{attribute 'linkalways'} 
{attribute 'no_explicit_call' := 'This FB is a CLASS and must be accessed using methods or properties'}
{attribute 'enable_dynamic_creation'}
FUNCTION_BLOCK _ETcVnDistanceType EXTENDS EnumDatatypeBase
VAR
	localData : ETcVnDistanceType;
	activeData : REFERENCE TO ETcVnDistanceType;
	enumBaseDatatype : _DINT(localData);
END_VAR

METHOD PRIVATE AddLocalEnumeration
VAR_INPUT
	Enumeration : T_MAXSTRING;
	Value : ETcVnDistanceType;
END_VAR
AddEnumeration(Enumeration, Value);
END_METHOD

PROPERTY PUBLIC Address : PVOID
GET
Address := ADR(activeData);
END_GET
END_PROPERTY

METHOD PUBLIC ClearReference
VAR_INPUT
END_VAR
activeData REF= localData;
SetBaseDatatypeReference();
END_METHOD

METHOD PUBLIC Clone : I_Datatype
VAR
    pClone : POINTER TO _ETcVnDistanceType;
END_VAR
pClone := __NEW(_ETcVnDistanceType(InitialValue := Value));
Clone := pClone^;
END_METHOD

METHOD FB_init : BOOL
VAR_INPUT
	bInitRetains : BOOL; // if TRUE, the retain variables are initialized (warm start / cold start)
	bInCopyCode : BOOL;  // if TRUE, the instance afterwards gets moved into the copy code (online change)
	InitialValue : ETcVnDistanceType;
END_VAR
localData := InitialValue;
AddBaseDatatype(enumBaseDatatype);
ClearReference();

AddLocalEnumeration('TCVN_DT_USER', ETcVnDistanceType.TCVN_DT_USER);
AddLocalEnumeration('TCVN_DT_L1', ETcVnDistanceType.TCVN_DT_L1);
AddLocalEnumeration('TCVN_DT_L2', ETcVnDistanceType.TCVN_DT_L2);
AddLocalEnumeration('TCVN_DT_C', ETcVnDistanceType.TCVN_DT_C);
AddLocalEnumeration('TCVN_DT_L12', ETcVnDistanceType.TCVN_DT_L12);
AddLocalEnumeration('TCVN_DT_FAIR', ETcVnDistanceType.TCVN_DT_FAIR);
AddLocalEnumeration('TCVN_DT_WELSCH', ETcVnDistanceType.TCVN_DT_WELSCH);
AddLocalEnumeration('TCVN_DT_HUBER ', ETcVnDistanceType.TCVN_DT_HUBER);
END_METHOD

PROPERTY PUBLIC Identifier : T_MAXSTRING
GET
Identifier := 'ETcVnDistanceType';
END_GET
END_PROPERTY

METHOD IsEnumeratorValueEqual : BOOL
VAR_INPUT
	Enumerator : I_KeyValueForwardEnumerator;
END_VAR
VAR
	storedValue : ETcVnDistanceType;
END_VAR
IF NOT Enumerator.TryGet(storedValue) THEN
	RETURN;
END_IF

IsEnumeratorValueEqual := storedValue = activeData;
END_METHOD

METHOD PUBLIC MakeReferenceTo
VAR_INPUT
	ReferenceTarget : REFERENCE TO ETcVnDistanceType;
END_VAR
activeData REF= ReferenceTarget;
SetBaseDatatypeReference();
END_METHOD

METHOD PROTECTED SetBaseDatatypeReference
VAR_INPUT
END_VAR
enumBaseDatatype.MakeReferenceTo(activeData);
END_METHOD

PROPERTY PUBLIC Size : UDINT
GET
Size := SIZEOF(activeData);
END_GET
END_PROPERTY

METHOD TryMakeReferenceTo : BOOL
VAR_INPUT
	Target : I_Datatype;
END_VAR
VAR
	targetAsEnum : I_EnumDatatype;
	pTargetData : POINTER TO ETcVnDistanceType;
END_VAR
IF NOT Target.TryResolveAsEnumDatatype(targetAsEnum) THEN
	RETURN;
END_IF

IF targetAsEnum.Identifier <> Identifier THEN
	RETURN;
END_IF

pTargetData := Target.Address;
activeData REF= pTargetData^;
SetBaseDatatypeReference();
TryMakeReferenceTo := TRUE;
END_METHOD

PROPERTY PUBLIC Value : ETcVnDistanceType
GET
Value := activeData;
END_GET
SET
activeData := Value;
END_SET
END_PROPERTY

END_FUNCTION_BLOCK

(* stored: Version 1.1.0.1
   POU _ETcVnDistanceType: Id {954cc886-1c48-4b8f-951f-ac6a83a2a936}, SpecialFunc None
   Folder Constructor: Id {fb5c8596-8fd6-4335-9b10-df8f59edb931}
   Folder Private: Id {43f32b86-f420-4c4a-aac4-444d1093c127}
   Folder Protected: Id {1a091fcb-0e9e-48fd-b72e-dbadfdf87a85}
   Method AddLocalEnumeration: Id {322149e7-12b9-41f5-82dd-626a557328c4}
   Property Address: Id {01a9870e-7d1d-4d5f-b29e-4366be6a689d}
   Get Get: Id {d20919d9-6241-4484-8b13-0e0121bc96c4}
   Method ClearReference: Id {58d30b87-4c4a-4012-a22a-db5281a453c4}
   Method Clone: Id {9af3a109-f29c-4016-b882-8b447552e10b}
   Method FB_init: Id {ee5fe9b0-6e39-485b-8810-c1a05e021a14}
   Property Identifier: Id {7bc38927-85bf-4f64-b89f-0889507db4f0}
   Get Get: Id {425772fa-6dfa-4c2c-bc2d-dbea81fe6e0b}
   Method IsEnumeratorValueEqual: Id {7c4c8e35-3811-43cd-901c-05199c54e8f4}
   Method MakeReferenceTo: Id {12f4b3f2-c244-4905-b295-492460ed57f5}
   Method SetBaseDatatypeReference: Id {2da79510-8cc9-449d-b118-477d00725754}
   Property Size: Id {71b73bbc-08e8-481c-888e-d36cf664227f}
   Get Get: Id {839c3150-3279-4a6c-92d0-946f13d1e4d8}
   Method TryMakeReferenceTo: Id {45856ae3-754b-4d98-bf24-bb53f3d2b1db}
   Property Value: Id {c76578a1-e29f-4acc-b42d-5113fcd9106e}
   Get Get: Id {97e00455-c944-44d1-a45e-09775be6c5b0}
   Set Set: Id {3ad7d7ce-c77d-435e-97dd-25ed1a9f5c58} *)
